FUNCTION ST08B_TO_BYTE
  (* Standard: 61499-1 *)
  (* Version 1.0, 2024-02-22, franz *)
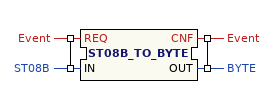
  EVENT_INPUT
    REQ WITH IN; (* Normal Execution Request *)
  END_EVENT
  EVENT_OUTPUT
    CNF WITH OUT; (* Execution Confirmation *)
  END_EVENT
  VAR_INPUT
    IN : ST08B; (* ST08B Input *)
  END_VAR
  VAR_OUTPUT
    OUT : BYTE; (* BYTE Output *)
  END_VAR
  BODY IN ST:
FUNCTION ST08B_TO_BYTE

VAR_INPUT
	IN : ST08B;    // ST08B Input
END_VAR

VAR_OUTPUT
	OUT : BYTE;    // BYTE Output
END_VAR

(* this Function extracts the 8 BOOLS from a byte *)
OUT.0 := IN.B_00;
OUT.1 := IN.B_01;
OUT.2 := IN.B_02;
OUT.3 := IN.B_03;
OUT.4 := IN.B_04;
OUT.5 := IN.B_05;
OUT.6 := IN.B_06;
OUT.7 := IN.B_07;

END_FUNCTION
  END_BODY
END_FUNCTION
